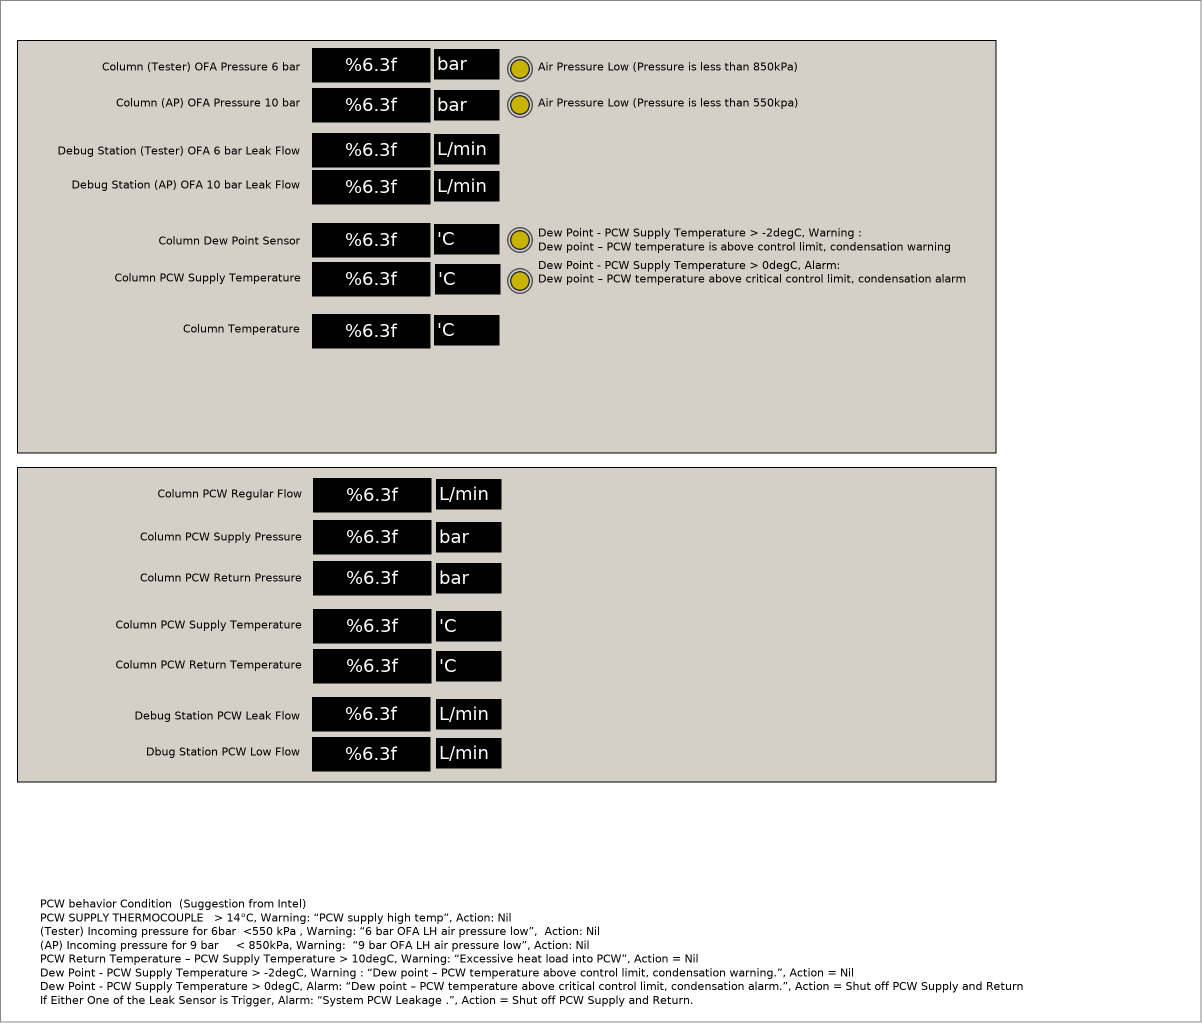
VISUALIZATION HMI_PCWBehaviour  // 1202x1023
    Rectangle (17,467 979x315)
    Rectangle (17,40 979x413)
    Textfield (311,47 120x36), "%6.3f", text variable: fbDebugColumn.stDebugColumnDIO.ipDBColumnTstAirPressure, input disabled if: TRUE
    Textfield (311,87 120x36), "%6.3f", text variable: fbDebugColumn.stDebugColumnDIO.ipDBColumnAPAirPressure, input disabled if: TRUE
    Textfield (311,132 120x36), "%6.3f", text variable: stDebugStation.fbDBStnSeq.stDebugStationDIO.ipDBStnTstAirLeakFlowSensor, input disabled if: TRUE
    Textfield (311,169 120x36), "%6.3f", text variable: stDebugStation.fbDBStnSeq.stDebugStationDIO.ipDBStnAPAirLeakFlowSensor, input disabled if: TRUE
    Label (42,136 261x30), "Debug Station (Tester) OFA 6 bar Leak Flow"
    Label (35,170 268x30), "Debug Station (AP) OFA 10 bar Leak Flow"
    Label (51,52 252x30), "Column (Tester) OFA Pressure 6 bar"
    Label (72,88 231x30), "Column (AP) OFA Pressure 10 bar"
    Textfield (311,696 120x36), "%6.3f", text variable: stDebugStation.fbDBStnSeq.stDebugStationDIO.ipDBStnPCWLeakFlowSensor, input disabled if: TRUE
    Textfield (311,736 120x36), "%6.3f", text variable: stDebugStation.fbDBStnSeq.stDebugStationDIO.ipDBStnPCWLowFlowSensor, input disabled if: TRUE
    Label (101,701 202x30), "Debug Station PCW Leak Flow"
    Label (55,737 248x30), "Dbug Station PCW Low Flow"
    Textfield (312,648 120x36), "%6.3f", text variable: fbDebugColumn.stDebugColumnDIO.ipDBColumnPCWReturnTemperature, input disabled if: TRUE
    Textfield (312,560 120x36), "%6.3f", text variable: fbDebugColumn.stDebugColumnDIO.ipDBColumnPCWReturnPressure, input disabled if: TRUE
    Textfield (312,477 120x36), "%6.3f", text variable: fbDebugColumn.stDebugColumnDIO.ipDBColumnPCWRegularFlowSensor, input disabled if: TRUE
    Textfield (312,519 120x36), "%6.3f", text variable: fbDebugColumn.stDebugColumnDIO.ipDBColumnPCWSupplyPressure, input disabled if: TRUE
    Textfield (312,608 120x36), "%6.3f", text variable: fbDebugColumn.stDebugColumnDIO.ipDBColumnPCWSupplyTemperature, input disabled if: TRUE
    Label (94,479 211x30), "Column PCW Regular Flow"
    Label (97,522 208x30), "Column PCW Supply Pressure"
    Label (122,563 183x30), "Column PCW Return Pressure"
    Label (76,610 229x30), "Column PCW Supply Temperature"
    Label (92,650 213x30), "Column PCW Return Temperature"
    Rectangle (436,479 65x30), "L/min"
    Rectangle (436,522 65x30), "bar"
    Rectangle (436,563 65x30), "bar"
    Rectangle (436,611 65x30), "'C"
    Rectangle (436,651 65x30), "'C"
    Rectangle (436,699 65x30), "L/min"
    Rectangle (436,738 65x30), "L/min"
    Rectangle (434,49 65x30), "bar"
    Rectangle (434,90 65x30), "bar"
    Rectangle (434,134 65x30), "L/min"
    Rectangle (434,171 65x30), "L/min"
    Textfield (311,222 120x36), "%6.3f", text variable: stDebugStation.fbDBStnSeq.stDebugStationDIO.ipDBStnTstAirLeakFlowSensor, input disabled if: TRUE
    Textfield (311,313 120x36), "%6.3f", text variable: fbDebugColumn.stDebugColumnDIO.ipDBColumnTempSensor, input disabled if: TRUE
    Label (124,226 179x30), "Column Dew Point Sensor"
    Label (153,314 150x30), "Column Temperature"
    Rectangle (434,224 65x30), "'C"
    Rectangle (434,315 65x30), "'C"
    Label (30,897 1170x124), "PCW behavior Condition (Suggestion from Intel) PCW SUPPLY THERMOCOUPLE > 14°C, Warning: “PCW supply high temp”, Action: Nil (Tester) Incoming pressure for 6bar <550 kPa , Warning: “6 bar OFA LH air pressure low”, Action: Nil (AP) Incoming pressure for 9 bar < 850kPa, Warning: “9 bar OFA LH air pressure low”, Action: Nil PCW Return Temperature – PCW Supply Temperature > 10degC, Warning: “Excessive heat load into PCW”, Action = Nil Dew Point - PCW Supply Temperature > -2degC, Warning : “Dew point – PCW temperature above control limit, condensation warning.”, Action = Nil Dew Point - PCW Supply Temperature > 0degC, Alarm: “Dew point – PCW temperature above critical control limit, condensation alarm.”, Action = Shut off PCW Supply and Return If Either One of the Leak Sensor is Trigger, Alarm: “System PCW Leakage .”, Action = Shut off PCW Supply and Return."
    Lamp1 (505,90 30x30), style: Lamp-Lamp1-Yellow
    Label (535,88 376x30), "Air Pressure Low (Pressure is less than 550kpa)"
    Lamp1 (505,54 30x30), style: Lamp-Lamp1-Yellow
    Label (535,52 376x30), "Air Pressure Low (Pressure is less than 850kPa)"
    Textfield (311,261 120x36), "%6.3f", text variable: fbDebugColumn.stDebugColumnDIO.ipDBColumnPCWSupplyTemperature, input disabled if: TRUE
    Label (75,263 229x30), "Column PCW Supply Temperature"
    Rectangle (435,264 65x30), "'C"
    Lamp1 (505,266 30x30), style: Lamp-Lamp1-Yellow
    Label (535,264 436x30), "Dew Point - PCW Supply Temperature > 0degC, Alarm: Dew point – PCW temperature above critical control limit, condensation alarm"
    Lamp1 (505,225 30x30), style: Lamp-Lamp1-Yellow
    Label (535,225 436x27), "Dew Point - PCW Supply Temperature > -2degC, Warning : Dew point – PCW temperature is above control limit, condensation warning"
END_VISUALIZATION

(* stored: Version 1.1.0.1, ProductVersion 3.1.4022.12
   Visu HMI_PCWBehaviour: Id {2ea90a57-c5e2-4750-b446-726b16a1e101} *)
